INTERFACE ISimulatable EXTENDS IObject

{attribute 'monitoring' := 'call'}
{attribute 'OPC.UA.DA' := '1'}
{attribute 'OPC.UA.DA.Access' := '1'}
PROPERTY FINAL SimulationMode : BOOL
GET
END_GET
END_PROPERTY

END_INTERFACE

(* stored: Version 1.1.0.1
   Itf ISimulatable: Id {64def839-9c7f-49fb-bb6c-6e139237e3fc}
   Property SimulationMode: Id {f5dfb847-33cc-4380-a1cf-0d2edbb1a6ef}
   Get Get: Id {26bbacea-8cbd-4c03-a1df-2721a1043836} *)
